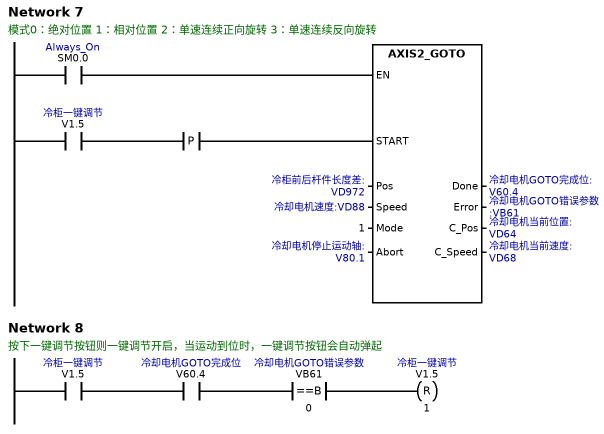
[picture p48: SBR18 networks 7-8]
Network 7
// 模式0：绝对位置 1：相对位置 2：单速连续正向旋转 3：单速连续反向旋转
LD     Always_On:SM0.0
=      L60.0
LD     冷柜一键调节:V1.5
EU
=      L63.7
LD     L60.0
CALL   AXIS2_GOTO:SBR12, L63.7, 冷柜前后杆件长度差:VD972, 冷却电机速度:VD88, 1, 冷却电机停止运动轴:V80.1, 冷却电机GOTO完成位:V60.4, 冷却电机GOTO错误参数:VB61, 冷却电机当前位置:VD64, 冷却电机当前速度:VD68
Network 8
// 按下一键调节按钮则一键调节开启，当运动到位时，一键调节按钮会自动弹起
LD     冷柜一键调节:V1.5
A      冷却电机GOTO完成位:V60.4
AB=    冷却电机GOTO错误参数:VB61, 0
R      冷柜一键调节:V1.5, 1
END_SUBROUTINE_BLOCK

SUBROUTINE_BLOCK 链传动电机控制:SBR19
TITLE=子程序注释
BEGIN
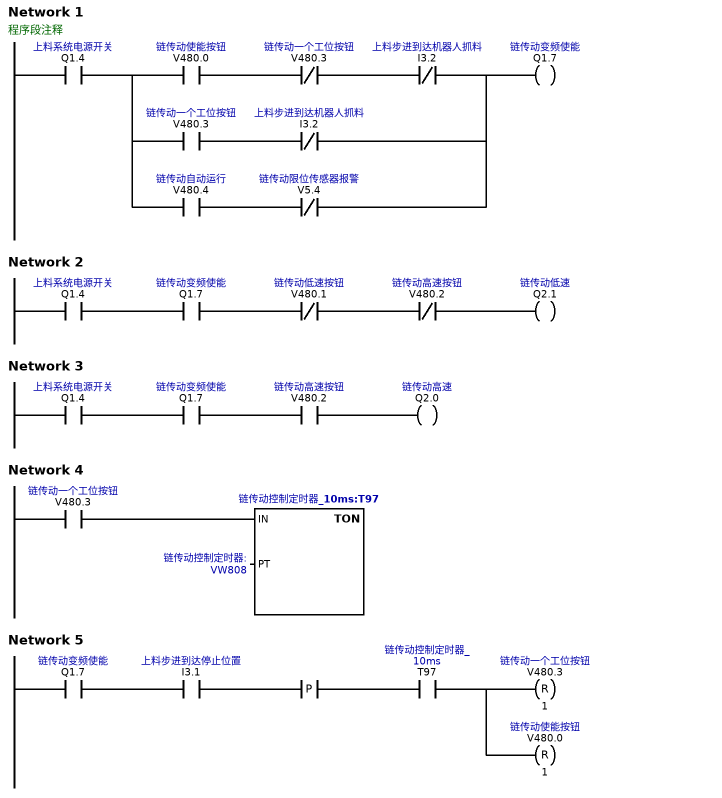
Network 1
// 程序段注释
LD     上料系统电源开关:Q1.4
LD     链传动使能按钮:V480.0
AN     链传动一个工位按钮:V480.3
AN     上料步进到达机器人抓料:I3.2
LD     链传动一个工位按钮:V480.3
AN     上料步进到达机器人抓料:I3.2
OLD
LD     链传动自动运行:V480.4
AN     链传动限位传感器报警:V5.4
OLD
ALD
=      链传动变频使能:Q1.7
Network 2
LD     上料系统电源开关:Q1.4
A      链传动变频使能:Q1.7
AN     链传动低速按钮:V480.1
AN     链传动高速按钮:V480.2
=      链传动低速:Q2.1
Network 3
LD     上料系统电源开关:Q1.4
A      链传动变频使能:Q1.7
A      链传动高速按钮:V480.2
=      链传动高速:Q2.0
Network 4
LD     链传动一个工位按钮:V480.3
TON    链传动控制定时器_10ms:T97, 链传动控制定时器:VW808
Network 5
LD     链传动变频使能:Q1.7
A      上料步进到达停止位置:I3.1
EU
A      链传动控制定时器_10ms:T97
R      链传动一个工位按钮:V480.3, 1
R      链传动使能按钮:V480.0, 1
END_SUBROUTINE_BLOCK

SUBROUTINE_BLOCK 数据初始化:SBR20
TITLE=子程序注释
BEGIN
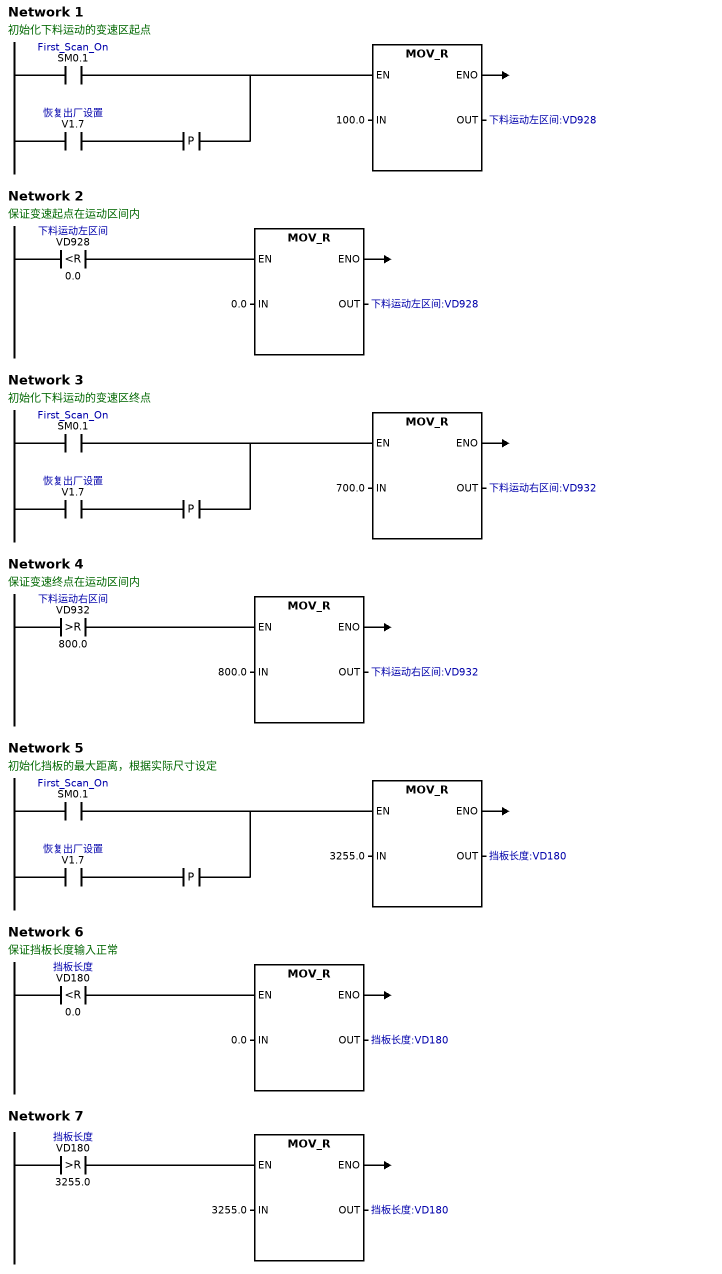
Network 1
// 初始化下料运动的变速区起点
LD     First_Scan_On:SM0.1
LD     恢复出厂设置:V1.7
EU
OLD
MOVR   100.0, 下料运动左区间:VD928
Network 2
// 保证变速起点在运动区间内
LDR<   下料运动左区间:VD928, 0.0
MOVR   0.0, 下料运动左区间:VD928
Network 3
// 初始化下料运动的变速区终点
LD     First_Scan_On:SM0.1
LD     恢复出厂设置:V1.7
EU
OLD
MOVR   700.0, 下料运动右区间:VD932
Network 4
// 保证变速终点在运动区间内
LDR>   下料运动右区间:VD932, 800.0
MOVR   800.0, 下料运动右区间:VD932
Network 5
// 初始化挡板的最大距离，根据实际尺寸设定
LD     First_Scan_On:SM0.1
LD     恢复出厂设置:V1.7
EU
OLD
MOVR   3255.0, 挡板长度:VD180
Network 6
// 保证挡板长度输入正常
LDR<   挡板长度:VD180, 0.0
MOVR   0.0, 挡板长度:VD180
Network 7
LDR>   挡板长度:VD180, 3255.0
MOVR   3255.0, 挡板长度:VD180
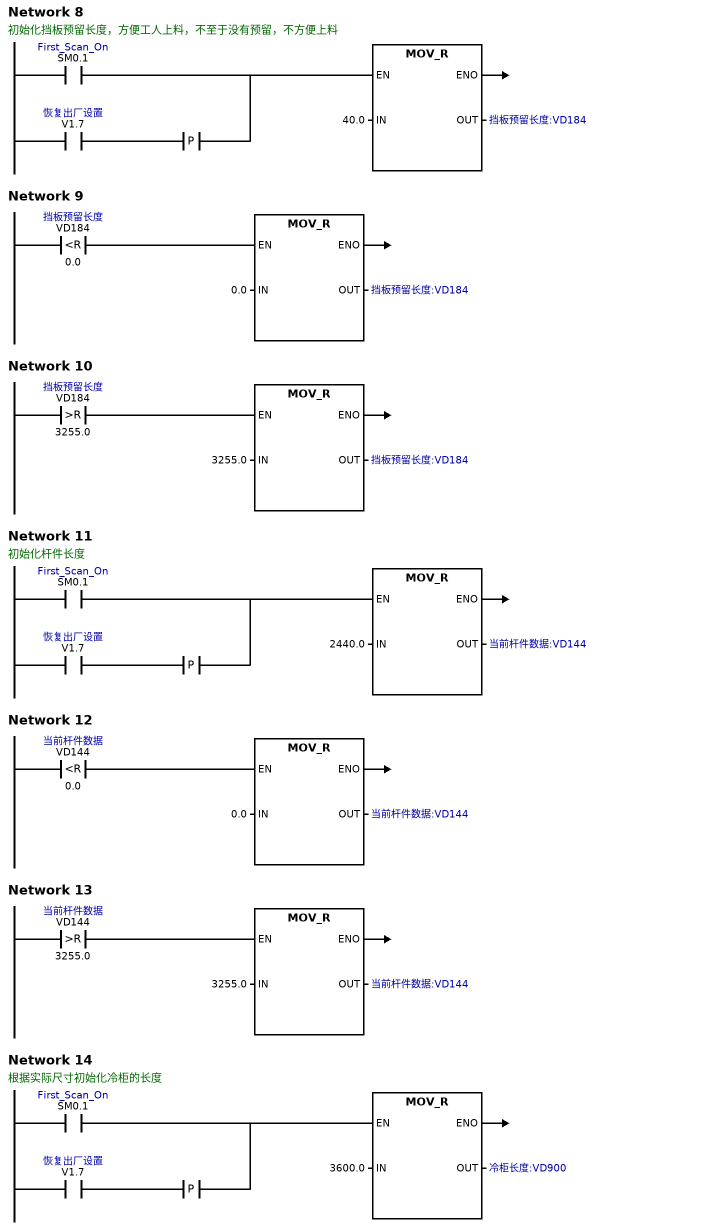
Network 8
// 初始化挡板预留长度，方便工人上料，不至于没有预留，不方便上料
LD     First_Scan_On:SM0.1
LD     恢复出厂设置:V1.7
EU
OLD
MOVR   40.0, 挡板预留长度:VD184
Network 9
LDR<   挡板预留长度:VD184, 0.0
MOVR   0.0, 挡板预留长度:VD184
Network 10
LDR>   挡板预留长度:VD184, 3255.0
MOVR   3255.0, 挡板预留长度:VD184
Network 11
// 初始化杆件长度
LD     First_Scan_On:SM0.1
LD     恢复出厂设置:V1.7
EU
OLD
MOVR   2440.0, 当前杆件数据:VD144
Network 12
LDR<   当前杆件数据:VD144, 0.0
MOVR   0.0, 当前杆件数据:VD144
Network 13
LDR>   当前杆件数据:VD144, 3255.0
MOVR   3255.0, 当前杆件数据:VD144
Network 14
// 根据实际尺寸初始化冷柜的长度
LD     First_Scan_On:SM0.1
LD     恢复出厂设置:V1.7
EU
OLD
MOVR   3600.0, 冷柜长度:VD900
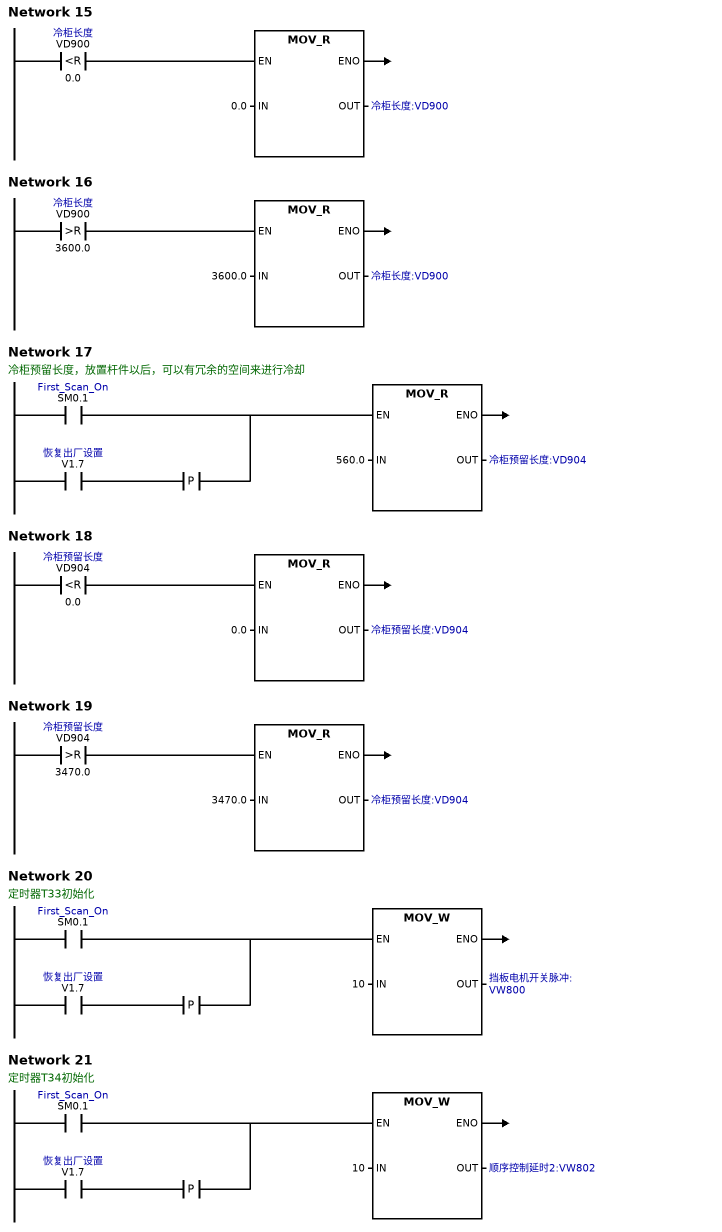
Network 15
LDR<   冷柜长度:VD900, 0.0
MOVR   0.0, 冷柜长度:VD900
Network 16
LDR>   冷柜长度:VD900, 3600.0
MOVR   3600.0, 冷柜长度:VD900
Network 17
// 冷柜预留长度，放置杆件以后，可以有冗余的空间来进行冷却
LD     First_Scan_On:SM0.1
LD     恢复出厂设置:V1.7
EU
OLD
MOVR   560.0, 冷柜预留长度:VD904
Network 18
LDR<   冷柜预留长度:VD904, 0.0
MOVR   0.0, 冷柜预留长度:VD904
Network 19
LDR>   冷柜预留长度:VD904, 3470.0
MOVR   3470.0, 冷柜预留长度:VD904
Network 20
// 定时器T33初始化
LD     First_Scan_On:SM0.1
LD     恢复出厂设置:V1.7
EU
OLD
MOVW   10, 挡板电机开关脉冲:VW800
Network 21
// 定时器T34初始化
LD     First_Scan_On:SM0.1
LD     恢复出厂设置:V1.7
EU
OLD
MOVW   10, 顺序控制延时2:VW802
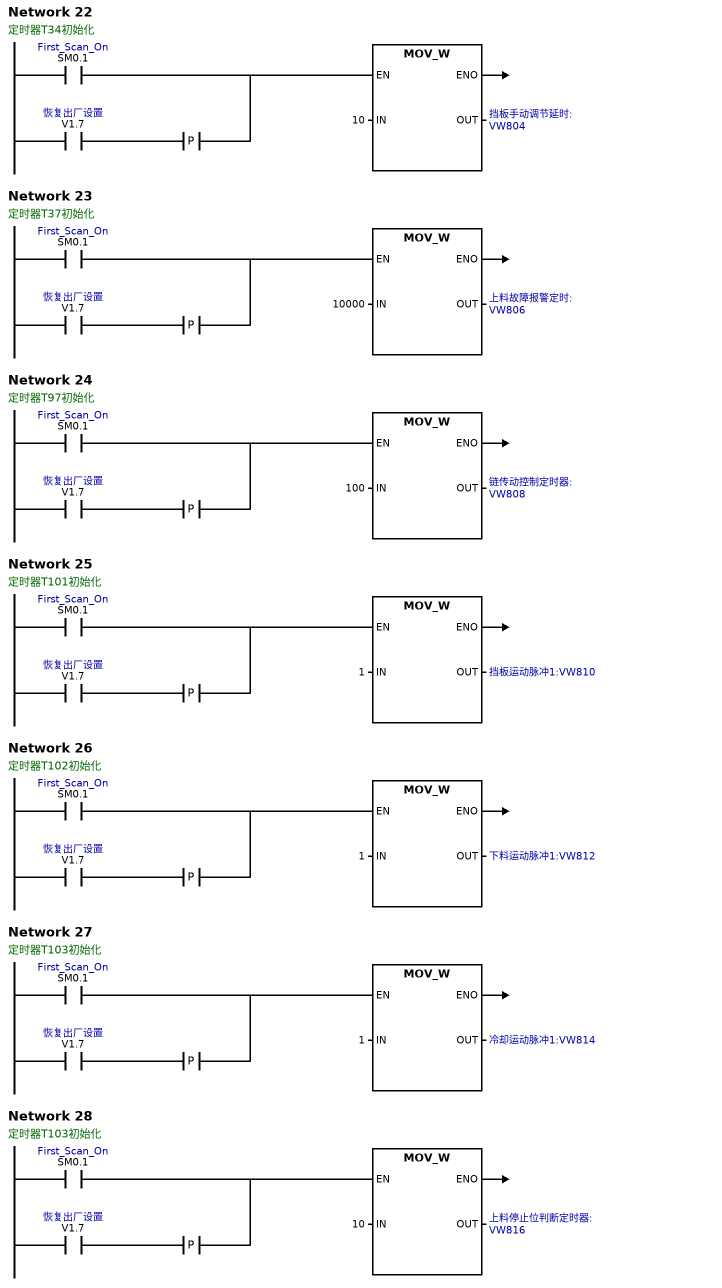
Network 22
// 定时器T34初始化
LD     First_Scan_On:SM0.1
LD     恢复出厂设置:V1.7
EU
OLD
MOVW   10, 挡板手动调节延时:VW804
Network 23
// 定时器T37初始化
LD     First_Scan_On:SM0.1
LD     恢复出厂设置:V1.7
EU
OLD
MOVW   10000, 上料故障报警定时:VW806
Network 24
// 定时器T97初始化
LD     First_Scan_On:SM0.1
LD     恢复出厂设置:V1.7
EU
OLD
MOVW   100, 链传动控制定时器:VW808
Network 25
// 定时器T101初始化
LD     First_Scan_On:SM0.1
LD     恢复出厂设置:V1.7
EU
OLD
MOVW   1, 挡板运动脉冲1:VW810
Network 26
// 定时器T102初始化
LD     First_Scan_On:SM0.1
LD     恢复出厂设置:V1.7
EU
OLD
MOVW   1, 下料运动脉冲1:VW812
Network 27
// 定时器T103初始化
LD     First_Scan_On:SM0.1
LD     恢复出厂设置:V1.7
EU
OLD
MOVW   1, 冷却运动脉冲1:VW814
Network 28
// 定时器T103初始化
LD     First_Scan_On:SM0.1
LD     恢复出厂设置:V1.7
EU
OLD
MOVW   10, 上料停止位判断定时器:VW816
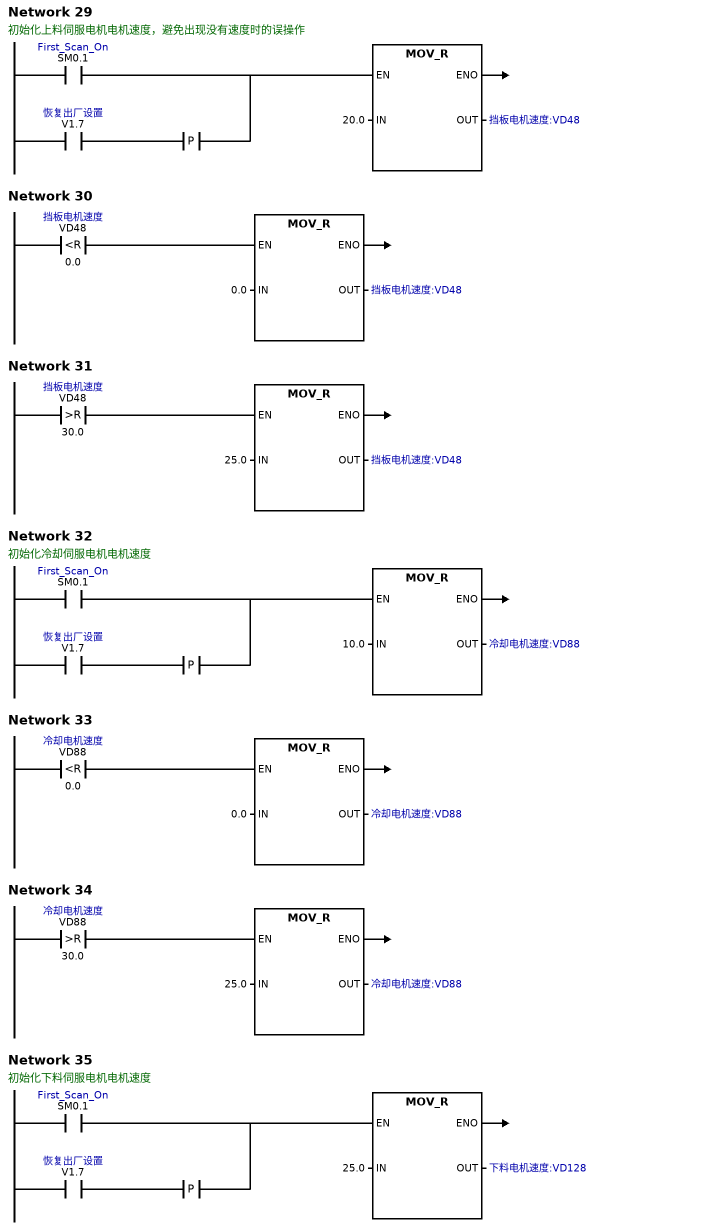
Network 29
// 初始化上料伺服电机电机速度，避免出现没有速度时的误操作
LD     First_Scan_On:SM0.1
LD     恢复出厂设置:V1.7
EU
OLD
MOVR   20.0, 挡板电机速度:VD48
Network 30
LDR<   挡板电机速度:VD48, 0.0
MOVR   0.0, 挡板电机速度:VD48
Network 31
LDR>   挡板电机速度:VD48, 30.0
MOVR   25.0, 挡板电机速度:VD48
Network 32
// 初始化冷却伺服电机电机速度
LD     First_Scan_On:SM0.1
LD     恢复出厂设置:V1.7
EU
OLD
MOVR   10.0, 冷却电机速度:VD88
Network 33
LDR<   冷却电机速度:VD88, 0.0
MOVR   0.0, 冷却电机速度:VD88
Network 34
LDR>   冷却电机速度:VD88, 30.0
MOVR   25.0, 冷却电机速度:VD88
Network 35
// 初始化下料伺服电机电机速度
LD     First_Scan_On:SM0.1
LD     恢复出厂设置:V1.7
EU
OLD
MOVR   25.0, 下料电机速度:VD128
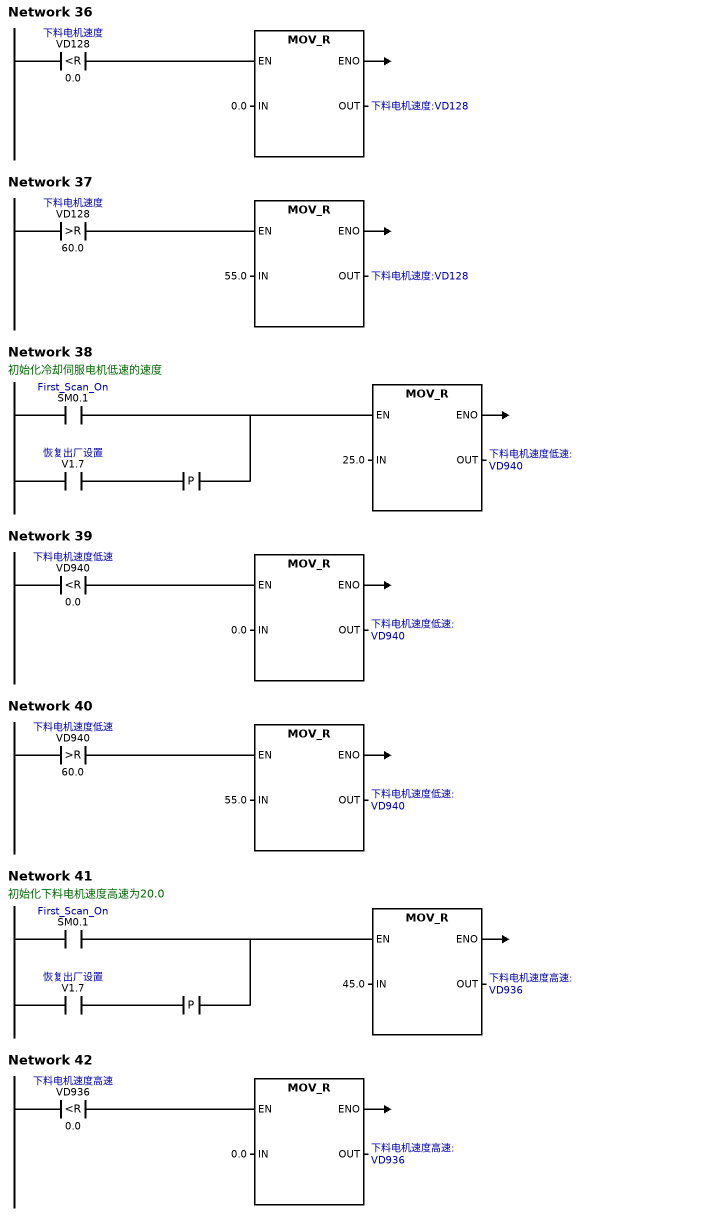
Network 36
LDR<   下料电机速度:VD128, 0.0
MOVR   0.0, 下料电机速度:VD128
Network 37
LDR>   下料电机速度:VD128, 60.0
MOVR   55.0, 下料电机速度:VD128
Network 38
// 初始化冷却伺服电机低速的速度
LD     First_Scan_On:SM0.1
LD     恢复出厂设置:V1.7
EU
OLD
MOVR   25.0, 下料电机速度低速:VD940
Network 39
LDR<   下料电机速度低速:VD940, 0.0
MOVR   0.0, 下料电机速度低速:VD940
Network 40
LDR>   下料电机速度低速:VD940, 60.0
MOVR   55.0, 下料电机速度低速:VD940
Network 41
// 初始化下料电机速度高速为20.0
LD     First_Scan_On:SM0.1
LD     恢复出厂设置:V1.7
EU
OLD
MOVR   45.0, 下料电机速度高速:VD936
Network 42
LDR<   下料电机速度高速:VD936, 0.0
MOVR   0.0, 下料电机速度高速:VD936
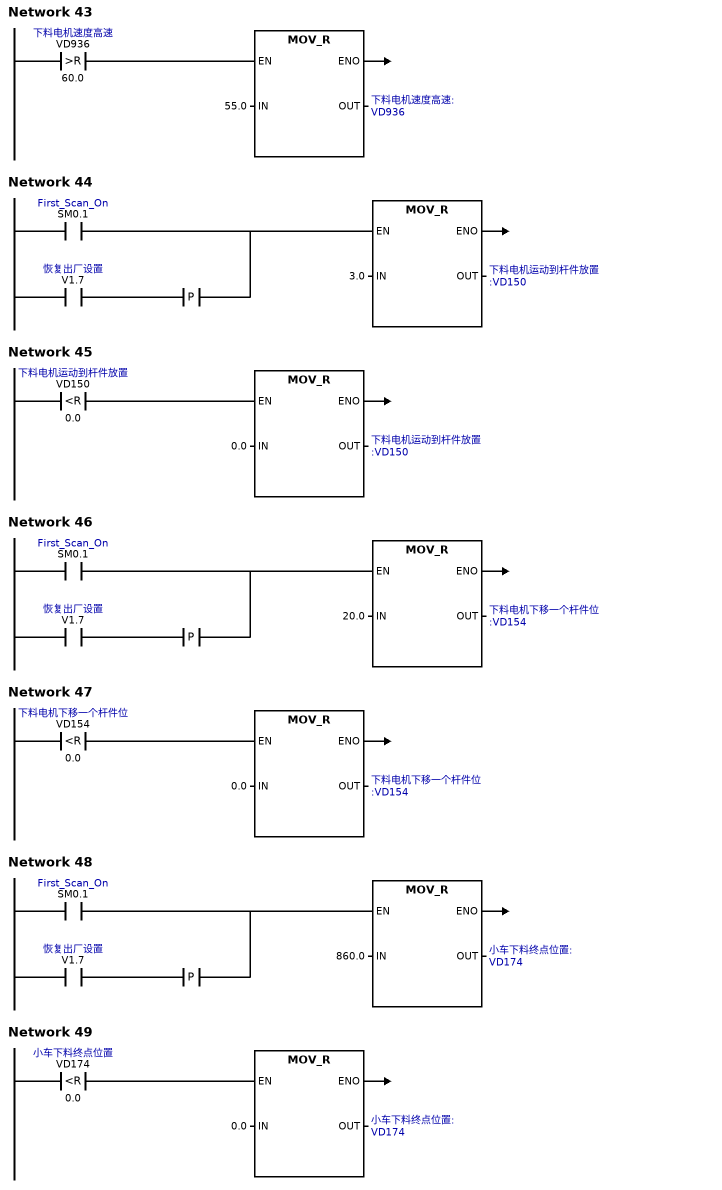
Network 43
LDR>   下料电机速度高速:VD936, 60.0
MOVR   55.0, 下料电机速度高速:VD936
Network 44
LD     First_Scan_On:SM0.1
LD     恢复出厂设置:V1.7
EU
OLD
MOVR   3.0, 下料电机运动到杆件放置:VD150
Network 45
LDR<   下料电机运动到杆件放置:VD150, 0.0
MOVR   0.0, 下料电机运动到杆件放置:VD150
Network 46
LD     First_Scan_On:SM0.1
LD     恢复出厂设置:V1.7
EU
OLD
MOVR   20.0, 下料电机下移一个杆件位:VD154
Network 47
LDR<   下料电机下移一个杆件位:VD154, 0.0
MOVR   0.0, 下料电机下移一个杆件位:VD154
Network 48
LD     First_Scan_On:SM0.1
LD     恢复出厂设置:V1.7
EU
OLD
MOVR   860.0, 小车下料终点位置:VD174
Network 49
LDR<   小车下料终点位置:VD174, 0.0
MOVR   0.0, 小车下料终点位置:VD174
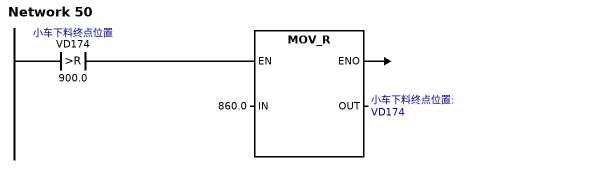
Network 50
LDR>   小车下料终点位置:VD174, 900.0
MOVR   860.0, 小车下料终点位置:VD174
END_SUBROUTINE_BLOCK

SUBROUTINE_BLOCK 故障报警:SBR21
TITLE=子程序注释
BEGIN
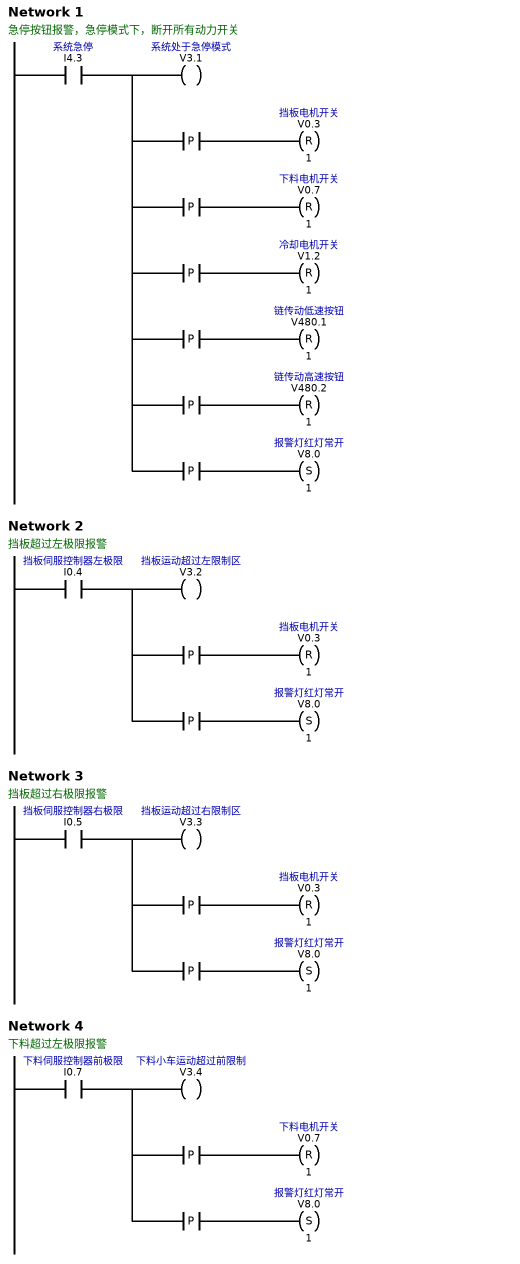
Network 1
// 急停按钮报警，急停模式下，断开所有动力开关
LD     系统急停:I4.3
LPS
=      系统处于急停模式:V3.1
EU
R      挡板电机开关:V0.3, 1
LRD
EU
R      下料电机开关:V0.7, 1
LRD
EU
R      冷却电机开关:V1.2, 1
LRD
EU
R      链传动低速按钮:V480.1, 1
LRD
EU
R      链传动高速按钮:V480.2, 1
LPP
EU
S      报警灯红灯常开:V8.0, 1
Network 2
// 挡板超过左极限报警
LD     挡板伺服控制器左极限:I0.4
LPS
=      挡板运动超过左限制区:V3.2
EU
R      挡板电机开关:V0.3, 1
LPP
EU
S      报警灯红灯常开:V8.0, 1
Network 3
// 挡板超过右极限报警
LD     挡板伺服控制器右极限:I0.5
LPS
=      挡板运动超过右限制区:V3.3
EU
R      挡板电机开关:V0.3, 1
LPP
EU
S      报警灯红灯常开:V8.0, 1
Network 4
// 下料超过左极限报警
LD     下料伺服控制器前极限:I0.7
LPS
=      下料小车运动超过前限制:V3.4
EU
R      下料电机开关:V0.7, 1
LPP
EU
S      报警灯红灯常开:V8.0, 1
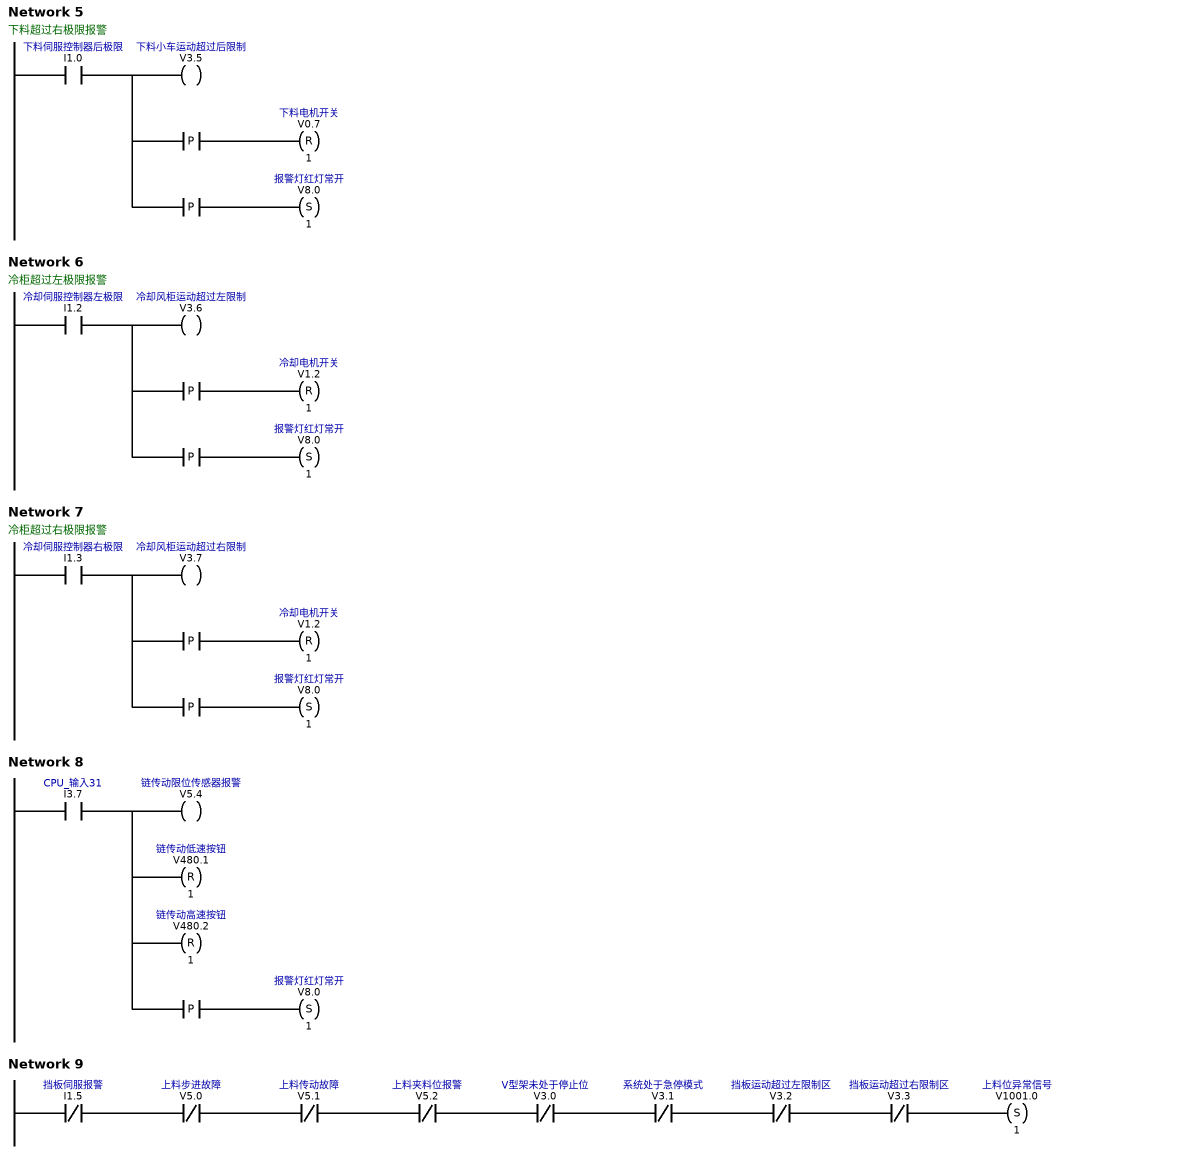
Network 5
// 下料超过右极限报警
LD     下料伺服控制器后极限:I1.0
LPS
=      下料小车运动超过后限制:V3.5
EU
R      下料电机开关:V0.7, 1
LPP
EU
S      报警灯红灯常开:V8.0, 1
Network 6
// 冷柜超过左极限报警
LD     冷却伺服控制器左极限:I1.2
LPS
=      冷却风柜运动超过左限制:V3.6
EU
R      冷却电机开关:V1.2, 1
LPP
EU
S      报警灯红灯常开:V8.0, 1
Network 7
// 冷柜超过右极限报警
LD     冷却伺服控制器右极限:I1.3
LPS
=      冷却风柜运动超过右限制:V3.7
EU
R      冷却电机开关:V1.2, 1
LPP
EU
S      报警灯红灯常开:V8.0, 1
Network 8
LD     CPU_输入31:I3.7
=      链传动限位传感器报警:V5.4
R      链传动低速按钮:V480.1, 1
R      链传动高速按钮:V480.2, 1
EU
S      报警灯红灯常开:V8.0, 1
Network 9
LDN    挡板伺服报警:I1.5
AN     上料步进故障:V5.0
AN     上料传动故障:V5.1
AN     上料夹料位报警:V5.2
AN     V型架未处于停止位:V3.0
AN     系统处于急停模式:V3.1
AN     挡板运动超过左限制区:V3.2
AN     挡板运动超过右限制区:V3.3
S      上料位异常信号:V1001.0, 1
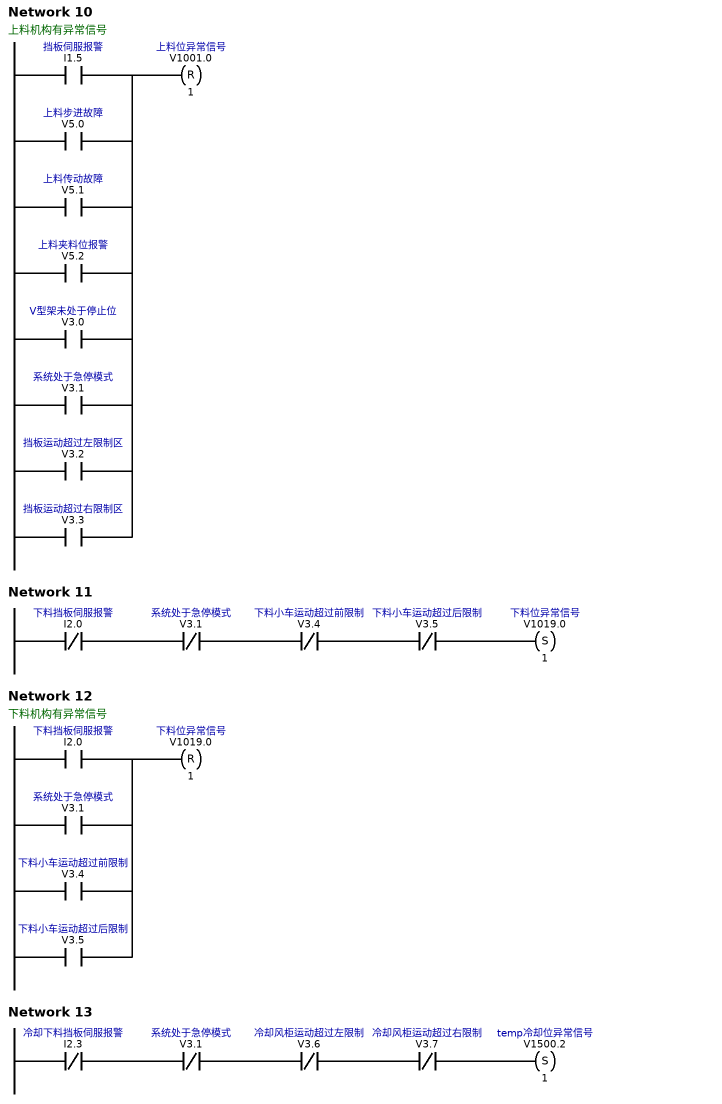
Network 10
// 上料机构有异常信号
LD     挡板伺服报警:I1.5
O      上料步进故障:V5.0
O      上料传动故障:V5.1
O      上料夹料位报警:V5.2
O      V型架未处于停止位:V3.0
O      系统处于急停模式:V3.1
O      挡板运动超过左限制区:V3.2
O      挡板运动超过右限制区:V3.3
R      上料位异常信号:V1001.0, 1
Network 11
LDN    下料挡板伺服报警:I2.0
AN     系统处于急停模式:V3.1
AN     下料小车运动超过前限制:V3.4
AN     下料小车运动超过后限制:V3.5
S      下料位异常信号:V1019.0, 1
Network 12
// 下料机构有异常信号
LD     下料挡板伺服报警:I2.0
O      系统处于急停模式:V3.1
O      下料小车运动超过前限制:V3.4
O      下料小车运动超过后限制:V3.5
R      下料位异常信号:V1019.0, 1
Network 13
LDN    冷却下料挡板伺服报警:I2.3
AN     系统处于急停模式:V3.1
AN     冷却风柜运动超过左限制:V3.6
AN     冷却风柜运动超过右限制:V3.7
S      temp冷却位异常信号:V1500.2, 1
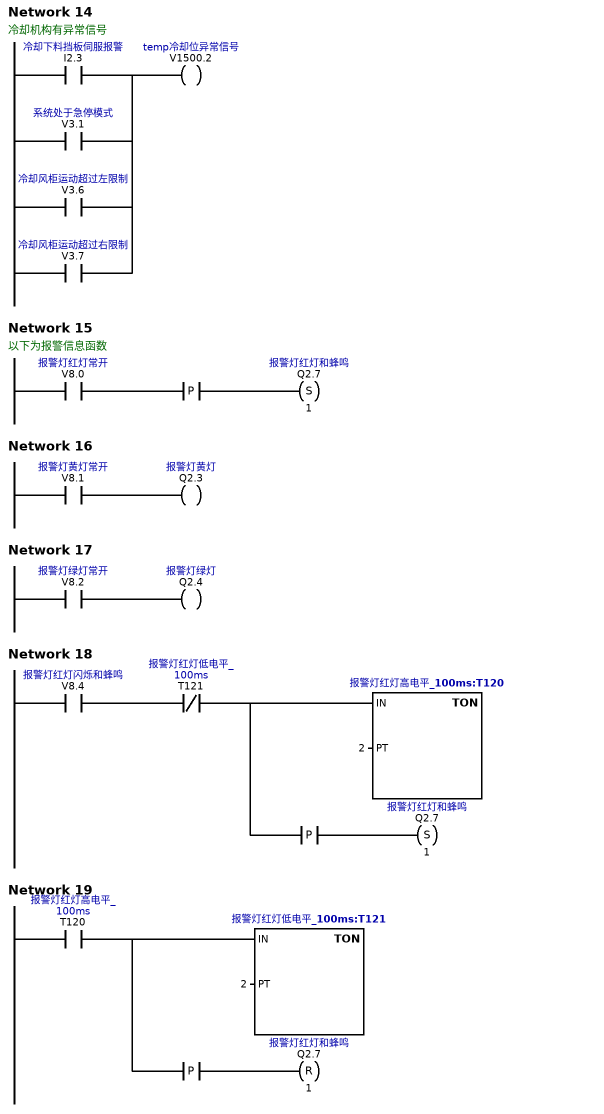
Network 14
// 冷却机构有异常信号
LD     冷却下料挡板伺服报警:I2.3
O      系统处于急停模式:V3.1
O      冷却风柜运动超过左限制:V3.6
O      冷却风柜运动超过右限制:V3.7
=      temp冷却位异常信号:V1500.2
Network 15
// 以下为报警信息函数
LD     报警灯红灯常开:V8.0
EU
S      报警灯红灯和蜂鸣:Q2.7, 1
Network 16
LD     报警灯黄灯常开:V8.1
=      报警灯黄灯:Q2.3
Network 17
LD     报警灯绿灯常开:V8.2
=      报警灯绿灯:Q2.4
Network 18
LD     报警灯红灯闪烁和蜂鸣:V8.4
AN     报警灯红灯低电平_100ms:T121
TON    报警灯红灯高电平_100ms:T120, 2
EU
S      报警灯红灯和蜂鸣:Q2.7, 1
Network 19
LD     报警灯红灯高电平_100ms:T120
TON    报警灯红灯低电平_100ms:T121, 2
EU
R      报警灯红灯和蜂鸣:Q2.7, 1
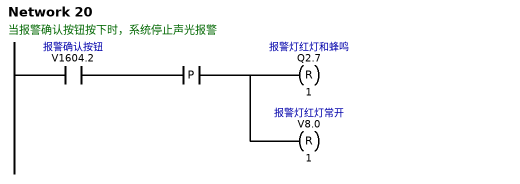
Network 20
// 当报警确认按钮按下时，系统停止声光报警
LD     报警确认按钮:V1604.2
EU
R      报警灯红灯和蜂鸣:Q2.7, 1
R      报警灯红灯常开:V8.0, 1
END_SUBROUTINE_BLOCK
